Yaskawa INFORM job: JERIKAN3.JBI

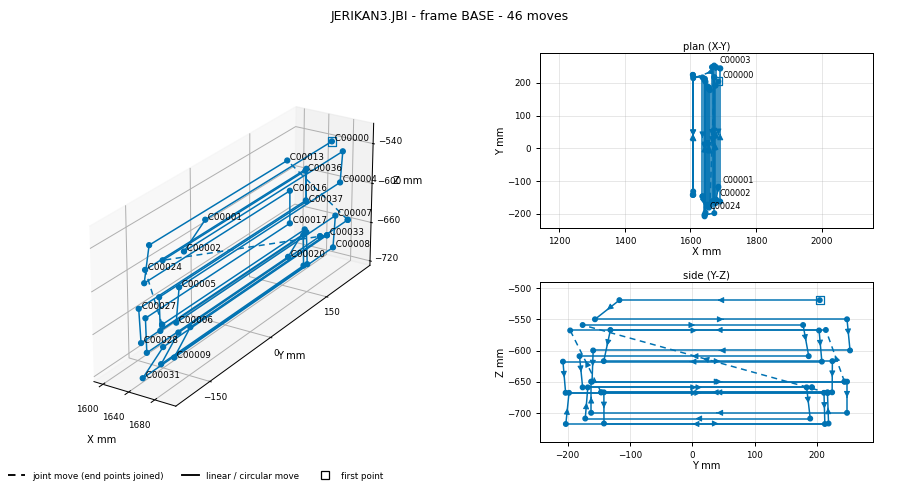
[picture p0: tool path of JERIKAN3.JBI in frame BASE, 46 of 52 moves have a stored position in this frame; points joined in program order, loops and branches not executed]
/JOB
//NAME JERIKAN3
//POS
///NPOS 46,0,46,0,0,0
///TOOL 0
///POSTYPE BASE
///RECTAN
///RCONF 1,0,0,0,0,0,0,0,0,0,0,0,0,0,0,0,0,0,0,0,0,0,0,0
C00000=1685.187728,204.218438,-519.027774,175.000000,-89.999999,5.000000
C00001=1685.187728,-117.082249,-519.027774,175.000000,-89.999999,5.000000
C00002=1678.371824,-156.249977,-549.712179,175.000000,-89.999999,5.000000
C00003=1678.371824,247.886578,-549.712179,175.000000,-89.999999,5.000000
C00004=1672.299350,252.738567,-599.712179,175.000000,-89.999999,5.000000
C00005=1672.299350,-159.132287,-599.712179,175.000000,-89.999999,5.000000
C00006=1668.421604,-160.959260,-649.712179,175.000000,-89.999999,5.000000
C00007=1668.421604,247.886578,-649.712179,175.000000,-89.999999,5.000000
C00008=1665.542578,247.886578,-699.712179,175.000000,-89.999999,5.000000
C00009=1665.542578,-162.367271,-699.712179,175.000000,-89.999999,5.000000
C00010=1690.840076,-162.367271,-649.712179,180.000000,-60.000000,0.000000
C00011=1690.840076,243.839307,-649.712179,180.000000,-60.000000,0.000000
C00012=1690.840076,243.839307,-649.712179,180.000000,-60.000000,0.000000
C00013=1608.386776,213.979694,-566.843652,175.000000,-89.999999,5.000000
C00014=1608.386776,-131.503496,-566.843652,175.000000,-89.999999,5.000000
C00015=1606.962140,-142.148327,-616.843652,175.000000,-89.999999,5.000000
C00016=1606.962140,224.430658,-616.843652,175.000000,-89.999999,5.000000
C00017=1607.694152,224.031189,-666.843652,175.000000,-89.999999,5.000000
C00018=1607.694152,-141.961716,-666.843652,175.000000,-89.999999,5.000000
C00019=1608.737370,-141.797724,-716.843652,175.000000,-89.999999,5.000000
C00020=1608.737370,218.313572,-716.843652,175.000000,-89.999999,5.000000
C00021=1636.682303,216.510519,-666.843652,180.000000,-60.000000,0.000000
C00022=1636.682303,-146.332938,-666.843652,180.000000,-60.000000,0.000000
C00023=1636.682303,-146.332938,-666.843652,180.000000,-60.000000,0.000000
C00024=1645.988188,-195.951034,-567.624198,175.000000,-89.999999,5.000000
C00025=1645.988188,203.098783,-567.624198,175.000000,-89.999999,5.000000
C00026=1643.151809,207.568799,-617.624198,175.000000,-89.999999,5.000000
C00027=1643.151809,-207.571342,-617.624198,175.000000,-89.999999,5.000000
C00028=1642.753786,-203.324967,-667.624198,175.000000,-89.999999,5.000000
C00029=1642.753786,210.962664,-667.624198,175.000000,-89.999999,5.000000
C00030=1643.962389,212.386850,-717.624198,175.000000,-89.999999,5.000000
C00031=1643.962389,-202.950442,-717.624198,175.000000,-89.999999,5.000000
C00032=1672.776655,-197.867365,-667.624198,180.000000,-60.000000,0.000000
C00033=1672.776655,216.914852,-667.624198,180.000000,-60.000000,0.000000
C00034=1672.776655,216.914852,-667.624198,180.000000,-60.000000,0.000000
C00035=1659.228245,-176.006884,-558.905595,175.000000,-89.999999,5.000000
C00036=1659.228245,177.469745,-558.905595,175.000000,-89.999999,5.000000
C00037=1656.375964,186.503362,-608.905595,175.000000,-89.999999,5.000000
C00038=1656.375964,-181.017961,-608.905595,175.000000,-89.999999,5.000000
C00039=1654.027607,-176.036172,-658.905595,175.000000,-89.999999,5.000000
C00040=1654.027607,183.156527,-658.905595,175.000000,-89.999999,5.000000
C00041=1651.566756,188.905939,-708.905595,175.000000,-89.999999,5.000000
C00042=1651.566756,-171.812884,-708.905595,175.000000,-89.999999,5.000000
C00043=1676.115400,-167.767938,-658.905595,180.000000,-60.000000,0.000000
C00044=1676.115400,191.579417,-658.905595,180.000000,-60.000000,0.000000
C00045=1676.115400,191.579417,-658.905595,180.000000,-60.000000,0.000000
///POSTYPE PULSE
///PULSE
EC00000=0
EC00001=0
EC00002=0
EC00003=0
EC00004=0
EC00005=0
EC00006=0
EC00007=0
EC00008=0
EC00009=0
EC00010=0
EC00011=0
EC00012=92160
EC00013=92160
EC00014=92160
EC00015=92160
EC00016=92160
EC00017=92160
EC00018=92160
EC00019=92160
EC00020=92160
EC00021=92160
EC00022=92160
EC00023=184320
EC00024=184320
EC00025=184320
EC00026=184320
EC00027=184320
EC00028=184320
EC00029=184320
EC00030=184320
EC00031=184320
EC00032=184320
EC00033=184320
EC00034=276480
EC00035=276480
EC00036=276480
EC00037=276480
EC00038=276480
EC00039=276480
EC00040=276480
EC00041=276480
EC00042=276480
EC00043=276480
EC00044=276480
EC00045=368640
//INST
///DATE 2023/02/08 10:58
///ATTR SC,RW,RJ
////FRAME BASE
///GROUP1 RB1,ST1
NOP
MOVJ P009 EX000 VJ=15.00
MOVJ P009 VJ=15.00
MOVJ C00000 EC00000 VJ=15.0
CALL JOB:SPYON
MOVL C00001 EC00001 V=150.0
MOVL C00002 EC00002 V=150.0
MOVL C00003 EC00003 V=150.0
MOVL C00004 EC00004 V=150.0
MOVL C00005 EC00005 V=150.0
MOVL C00006 EC00006 V=150.0
MOVL C00007 EC00007 V=150.0
MOVL C00008 EC00008 V=150.0
MOVL C00009 EC00009 V=150.0
MOVL C00010 EC00010 V=150.0
MOVL C00011 EC00011 V=150.0
CALL JOB:SPYOF
MOVJ P009 VJ=15.00
MOVL C00012 EC00012 V=150.0
MOVJ C00013 EC00013 VJ=15.0
CALL JOB:SPYON
MOVL C00014 EC00014 V=150.0
MOVL C00015 EC00015 V=150.0
MOVL C00016 EC00016 V=150.0
MOVL C00017 EC00017 V=150.0
MOVL C00018 EC00018 V=150.0
MOVL C00019 EC00019 V=150.0
MOVL C00020 EC00020 V=150.0
MOVL C00021 EC00021 V=150.0
MOVL C00022 EC00022 V=150.0
CALL JOB:SPYOF
MOVJ P009 VJ=15.00
MOVL C00023 EC00023 V=150.0
MOVJ C00024 EC00024 VJ=15.0
CALL JOB:SPYON
MOVL C00025 EC00025 V=150.0
MOVL C00026 EC00026 V=150.0
MOVL C00027 EC00027 V=150.0
MOVL C00028 EC00028 V=150.0
MOVL C00029 EC00029 V=150.0
MOVL C00030 EC00030 V=150.0
MOVL C00031 EC00031 V=150.0
MOVL C00032 EC00032 V=150.0
MOVL C00033 EC00033 V=150.0
CALL JOB:SPYOF
MOVJ P009 VJ=15.00
MOVL C00034 EC00034 V=150.0
MOVJ C00035 EC00035 VJ=15.0
CALL JOB:SPYON
MOVL C00036 EC00036 V=150.0
MOVL C00037 EC00037 V=150.0
MOVL C00038 EC00038 V=150.0
MOVL C00039 EC00039 V=150.0
MOVL C00040 EC00040 V=150.0
MOVL C00041 EC00041 V=150.0
MOVL C00042 EC00042 V=150.0
MOVL C00043 EC00043 V=150.0
MOVL C00044 EC00044 V=150.0
CALL JOB:SPYOF
MOVJ P009 VJ=15.00
MOVL C00045 EC00045 V=150.0
END
